(*~
<docu>
<summary>
	Provides a mechanism for inspecting status of discrete signal.	
</summary>
</docu>
~*)
FUNCTION_BLOCK TcoAnalogueInspector EXTENDS TcoInspector
VAR
    _data : TcoAnalogueInspectorData;
	{attribute 'hide'}
	_lastOutValue : LREAL;
END_VAR

(*~
<docu>
<summary>
	Gets data of this inspector.
</summary>
</docu>
~*)
PROPERTY Data : REFERENCE TO TcoAnalogueInspectorData
GET
Data REF= _data;
END_GET
END_PROPERTY

(*~
<docu>
<summary>
	Inspects the signal and evaluates that it matches the value set in `RequiredStatus`.
</summary>
<returns>
	Returns the interface with information about the state of inspection.
</returns>
</docu>
~*)
METHOD Inspect : IInspector
VAR_INPUT
    Status : LREAL;
END_VAR

VAR
	tmpResult : BOOL;
	_minimum : LREAL;
	_value : LREAL;
	_maximum : LREAL;
	_lastOutValue : LREAL;
END_VAR

VAR CONSTANT
    epsilon : REAL := 100000;
END_VAR
Inspect := THIS^;

OnEnterInspection();

_inspectionData REF= _data;

Invoke();

IF (Execute()) THEN
    IF (_data.IsByPassed) THEN
        _data.Result    := eInspectorResult.Bypassed;
        _data.TimeStamp := Context.RealTimeClock.NowLocal();
        DoneWhen(TRUE);
        RETURN;
    END_IF

	_data.Result := eInspectorResult.Running;
	
	_minimum := (Data.RequiredMin * epsilon);
	_value := (Status * epsilon);
	_maximum := (Data.RequiredMax * epsilon);
	
     Data.DetectedStatus := Status;
	
	 tmpResult := (_minimum <= _value) AND (_maximum >= _value);
		
	 IF(NOT tmpResult) THEN
		_lastOutValue := Status;
	  END_IF
		
	 _failTimer(IN := TRUE, PT := _data.FailTime);
     _passTimer(IN := tmpResult, PT := _data.PassTime);
		  
     DoneWhen(_failTimer.Q OR _passTimer.Q);
END_IF;
END_METHOD

(*~
	<docu>
		<summary>
			Executes when task reaches the ```Done``` state .
		</summary>			
	</docu>	
~*)
METHOD PROTECTED OnDone
SUPER^.OnDone();
IF (_data.Result = eInspectorResult.Failed) THEN
     _data.DetectedStatus := _lastOutValue;
END_IF
END_METHOD

END_FUNCTION_BLOCK

(* stored: Version 1.1.0.1, ProductVersion 3.1.4024.9
   POU TcoAnalogueInspector: Id {ed836f0b-3319-05d9-1710-05ac209c74d2}, SpecialFunc None
   Property Data: Id {130749e8-fcf6-0744-3fe0-87dc486f505f}
   Get Get: Id {526cbef3-3b72-0ac9-38bd-c119084cf8c0}
   Method Inspect: Id {c118bb5d-5c06-0c92-0167-b09658df5a96}
   Method OnDone: Id {bb771705-c5a7-01ce-0fed-8852b88b3c08} *)
